// TIA Portal V17 export
// export: Created 2023-03-24T09:45:04.5136241Z, ExportSetting None, DisplayName Totally Integrated Automation Portal, DisplayVersion V17 Update 4, DisplayName TIA Portal Openness, DisplayVersion V17 Update 4, DisplayName TIA Portal Version Control Interface, DisplayVersion V17, DisplayName STEP 7 Professional, DisplayVersion V17 Update 4, DisplayName STEP 7 Safety, DisplayVersion V17, DisplayName WinCC Advanced / Unified PC, DisplayVersion V17 Update 4
FUNCTION "FC_DI" : Void   // FC12, LAD
TITLE = FC_DI
{ S7_Optimized_Access := 'FALSE' }
// Digital Input
// stored: SetENOAutomatically false
BEGIN

REGION Network 1: CONTROL VIA HW INTERFACE
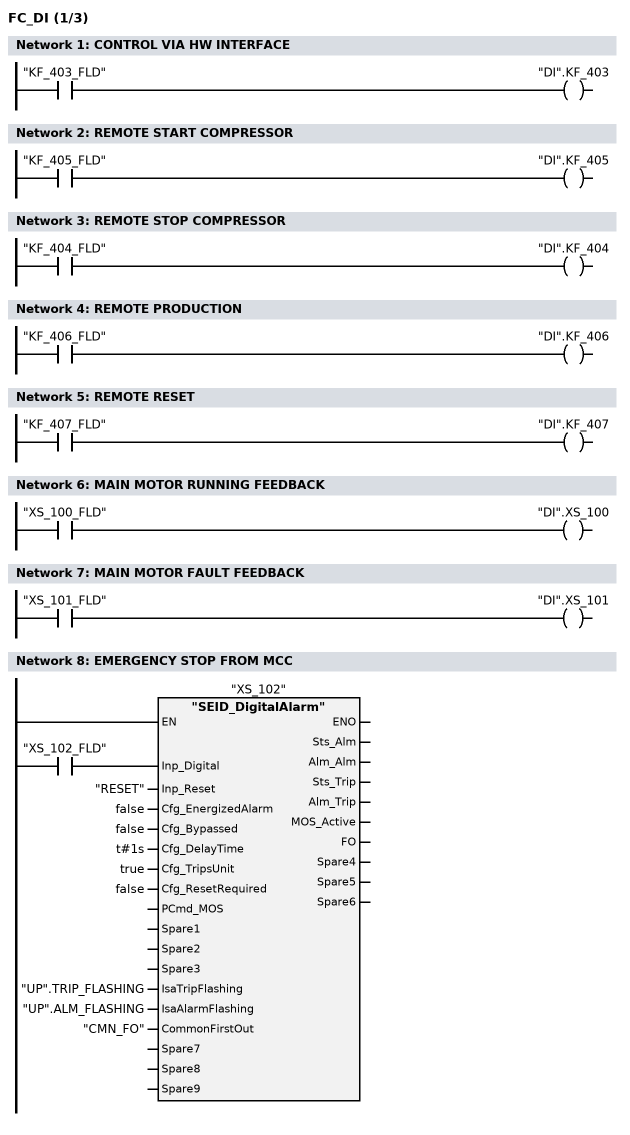
   RUNG wire#powerrail
      Contact( "KF_403_FLD" )
      Coil( "DI".KF_403 )
   END_RUNG
   // the same network as SCL:
   "DI".KF_403 := "KF_403_FLD";
END_REGION

REGION Network 2: REMOTE START COMPRESSOR
   RUNG wire#powerrail
      Contact( "KF_405_FLD" )
      Coil( "DI".KF_405 )
   END_RUNG
   // the same network as SCL:
   "DI".KF_405 := "KF_405_FLD";
END_REGION

REGION Network 3: REMOTE STOP COMPRESSOR
   RUNG wire#powerrail
      Contact( "KF_404_FLD" )
      Coil( "DI".KF_404 )
   END_RUNG
   // the same network as SCL:
   "DI".KF_404 := "KF_404_FLD";
END_REGION

REGION Network 4: REMOTE PRODUCTION
   RUNG wire#powerrail
      Contact( "KF_406_FLD" )
      Coil( "DI".KF_406 )
   END_RUNG
   // the same network as SCL:
   "DI".KF_406 := "KF_406_FLD";
END_REGION

REGION Network 5: REMOTE RESET
   RUNG wire#powerrail
      Contact( "KF_407_FLD" )
      Coil( "DI".KF_407 )
   END_RUNG
   // the same network as SCL:
   "DI".KF_407 := "KF_407_FLD";
END_REGION

REGION Network 6: MAIN MOTOR RUNNING FEEDBACK
   RUNG wire#powerrail
      Contact( "XS_100_FLD" )
      Coil( "DI".XS_100 )
   END_RUNG
   // the same network as SCL:
   "DI".XS_100 := "XS_100_FLD";
END_REGION

REGION Network 7: MAIN MOTOR FAULT FEEDBACK
   RUNG wire#powerrail
      Contact( "XS_101_FLD" )
      Coil( "DI".XS_101 )
   END_RUNG
   // the same network as SCL:
   "DI".XS_101 := "XS_101_FLD";
END_REGION

REGION Network 8: EMERGENCY STOP FROM MCC
   RUNG wire#powerrail
      "XS_102"(Inp_Digital := wire#w1, Inp_Reset := "RESET", Cfg_EnergizedAlarm := false, Cfg_Bypassed := false, Cfg_DelayTime := t#1s, Cfg_TripsUnit := true, Cfg_ResetRequired := false, PCmd_MOS :=, Spare1 :=, Spare2 :=, Spare3 :=, IsaTripFlashing := "UP".TRIP_FLASHING, IsaAlarmFlashing := "UP".ALM_FLASHING, CommonFirstOut := "CMN_FO", Spare7 :=, Spare8 :=, Spare9 :=, Sts_Alm =>, Alm_Alm =>, Sts_Trip =>, Alm_Trip =>, MOS_Active =>, FO =>, Spare4 =>, Spare5 =>, Spare6 =>)
   END_RUNG
   RUNG wire#powerrail
      Contact( "XS_102_FLD" )
   END_RUNG wire#w1
   // the same network as SCL:
   "XS_102"(Inp_Digital := "XS_102_FLD",   // "SEID_DigitalAlarm"
            Inp_Reset := "RESET",
            Cfg_EnergizedAlarm := false,
            Cfg_Bypassed := false,
            Cfg_DelayTime := t#1s,
            Cfg_TripsUnit := true,
            Cfg_ResetRequired := false,
            IsaTripFlashing := "UP".TRIP_FLASHING,
            IsaAlarmFlashing := "UP".ALM_FLASHING,
            CommonFirstOut := "CMN_FO");
END_REGION

REGION Network 9: HIGH TEMPERATURE FROM MCC
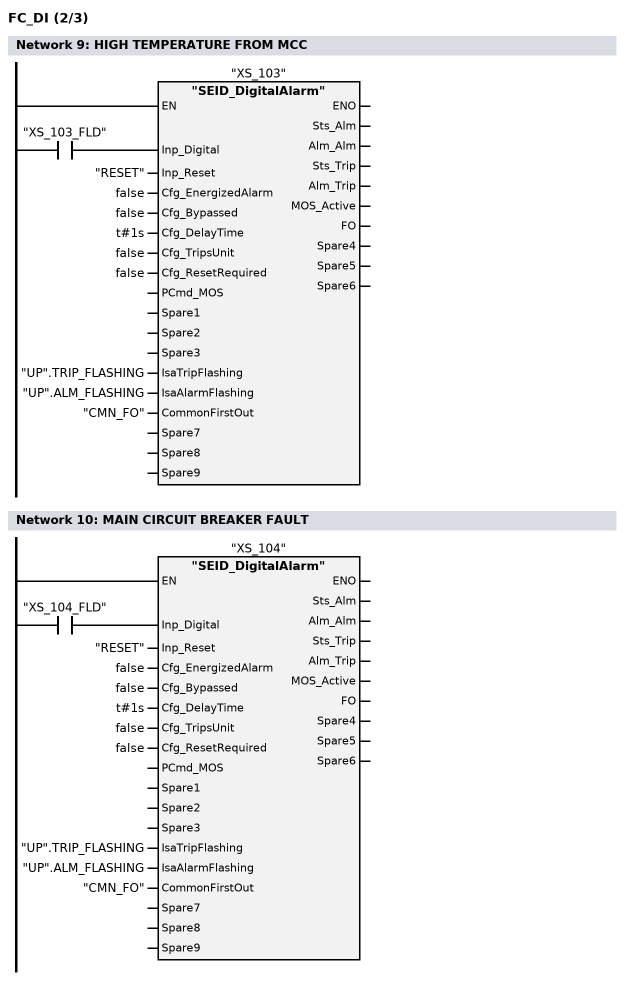
   RUNG wire#powerrail
      "XS_103"(Inp_Digital := wire#w1, Inp_Reset := "RESET", Cfg_EnergizedAlarm := false, Cfg_Bypassed := false, Cfg_DelayTime := t#1s, Cfg_TripsUnit := false, Cfg_ResetRequired := false, PCmd_MOS :=, Spare1 :=, Spare2 :=, Spare3 :=, IsaTripFlashing := "UP".TRIP_FLASHING, IsaAlarmFlashing := "UP".ALM_FLASHING, CommonFirstOut := "CMN_FO", Spare7 :=, Spare8 :=, Spare9 :=, Sts_Alm =>, Alm_Alm =>, Sts_Trip =>, Alm_Trip =>, MOS_Active =>, FO =>, Spare4 =>, Spare5 =>, Spare6 =>)
   END_RUNG
   RUNG wire#powerrail
      Contact( "XS_103_FLD" )
   END_RUNG wire#w1
   // the same network as SCL:
   "XS_103"(Inp_Digital := "XS_103_FLD",   // "SEID_DigitalAlarm"
            Inp_Reset := "RESET",
            Cfg_EnergizedAlarm := false,
            Cfg_Bypassed := false,
            Cfg_DelayTime := t#1s,
            Cfg_TripsUnit := false,
            Cfg_ResetRequired := false,
            IsaTripFlashing := "UP".TRIP_FLASHING,
            IsaAlarmFlashing := "UP".ALM_FLASHING,
            CommonFirstOut := "CMN_FO");
END_REGION

REGION Network 10: MAIN CIRCUIT BREAKER FAULT
   RUNG wire#powerrail
      "XS_104"(Inp_Digital := wire#w1, Inp_Reset := "RESET", Cfg_EnergizedAlarm := false, Cfg_Bypassed := false, Cfg_DelayTime := t#1s, Cfg_TripsUnit := false, Cfg_ResetRequired := false, PCmd_MOS :=, Spare1 :=, Spare2 :=, Spare3 :=, IsaTripFlashing := "UP".TRIP_FLASHING, IsaAlarmFlashing := "UP".ALM_FLASHING, CommonFirstOut := "CMN_FO", Spare7 :=, Spare8 :=, Spare9 :=, Sts_Alm =>, Alm_Alm =>, Sts_Trip =>, Alm_Trip =>, MOS_Active =>, FO =>, Spare4 =>, Spare5 =>, Spare6 =>)
   END_RUNG
   RUNG wire#powerrail
      Contact( "XS_104_FLD" )
   END_RUNG wire#w1
   // the same network as SCL:
   "XS_104"(Inp_Digital := "XS_104_FLD",   // "SEID_DigitalAlarm"
            Inp_Reset := "RESET",
            Cfg_EnergizedAlarm := false,
            Cfg_Bypassed := false,
            Cfg_DelayTime := t#1s,
            Cfg_TripsUnit := false,
            Cfg_ResetRequired := false,
            IsaTripFlashing := "UP".TRIP_FLASHING,
            IsaAlarmFlashing := "UP".ALM_FLASHING,
            CommonFirstOut := "CMN_FO");
END_REGION

REGION Network 11: UCP INTERNAL HIGH TEMPERATURE
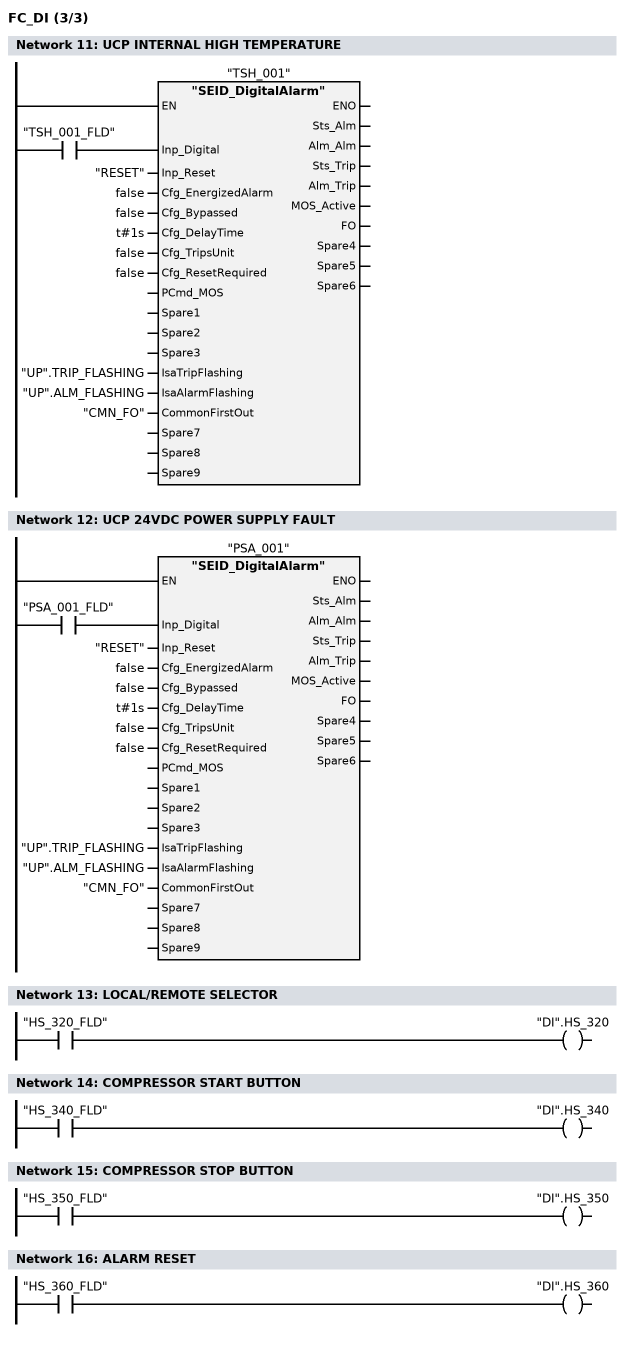
   RUNG wire#powerrail
      "TSH_001"(Inp_Digital := wire#w1, Inp_Reset := "RESET", Cfg_EnergizedAlarm := false, Cfg_Bypassed := false, Cfg_DelayTime := t#1s, Cfg_TripsUnit := false, Cfg_ResetRequired := false, PCmd_MOS :=, Spare1 :=, Spare2 :=, Spare3 :=, IsaTripFlashing := "UP".TRIP_FLASHING, IsaAlarmFlashing := "UP".ALM_FLASHING, CommonFirstOut := "CMN_FO", Spare7 :=, Spare8 :=, Spare9 :=, Sts_Alm =>, Alm_Alm =>, Sts_Trip =>, Alm_Trip =>, MOS_Active =>, FO =>, Spare4 =>, Spare5 =>, Spare6 =>)
   END_RUNG
   RUNG wire#powerrail
      Contact( "TSH_001_FLD" )
   END_RUNG wire#w1
   // the same network as SCL:
   "TSH_001"(Inp_Digital := "TSH_001_FLD",   // "SEID_DigitalAlarm"
             Inp_Reset := "RESET",
             Cfg_EnergizedAlarm := false,
             Cfg_Bypassed := false,
             Cfg_DelayTime := t#1s,
             Cfg_TripsUnit := false,
             Cfg_ResetRequired := false,
             IsaTripFlashing := "UP".TRIP_FLASHING,
             IsaAlarmFlashing := "UP".ALM_FLASHING,
             CommonFirstOut := "CMN_FO");
END_REGION

REGION Network 12: UCP 24VDC POWER SUPPLY FAULT
   RUNG wire#powerrail
      "PSA_001"(Inp_Digital := wire#w1, Inp_Reset := "RESET", Cfg_EnergizedAlarm := false, Cfg_Bypassed := false, Cfg_DelayTime := t#1s, Cfg_TripsUnit := false, Cfg_ResetRequired := false, PCmd_MOS :=, Spare1 :=, Spare2 :=, Spare3 :=, IsaTripFlashing := "UP".TRIP_FLASHING, IsaAlarmFlashing := "UP".ALM_FLASHING, CommonFirstOut := "CMN_FO", Spare7 :=, Spare8 :=, Spare9 :=, Sts_Alm =>, Alm_Alm =>, Sts_Trip =>, Alm_Trip =>, MOS_Active =>, FO =>, Spare4 =>, Spare5 =>, Spare6 =>)
   END_RUNG
   RUNG wire#powerrail
      Contact( "PSA_001_FLD" )
   END_RUNG wire#w1
   // the same network as SCL:
   "PSA_001"(Inp_Digital := "PSA_001_FLD",   // "SEID_DigitalAlarm"
             Inp_Reset := "RESET",
             Cfg_EnergizedAlarm := false,
             Cfg_Bypassed := false,
             Cfg_DelayTime := t#1s,
             Cfg_TripsUnit := false,
             Cfg_ResetRequired := false,
             IsaTripFlashing := "UP".TRIP_FLASHING,
             IsaAlarmFlashing := "UP".ALM_FLASHING,
             CommonFirstOut := "CMN_FO");
END_REGION

REGION Network 13: LOCAL/REMOTE SELECTOR
   RUNG wire#powerrail
      Contact( "HS_320_FLD" )
      Coil( "DI".HS_320 )
   END_RUNG
   // the same network as SCL:
   "DI".HS_320 := "HS_320_FLD";
END_REGION

REGION Network 14: COMPRESSOR START BUTTON
   RUNG wire#powerrail
      Contact( "HS_340_FLD" )
      Coil( "DI".HS_340 )
   END_RUNG
   // the same network as SCL:
   "DI".HS_340 := "HS_340_FLD";
END_REGION

REGION Network 15: COMPRESSOR STOP BUTTON
   RUNG wire#powerrail
      Contact( "HS_350_FLD" )
      Coil( "DI".HS_350 )
   END_RUNG
   // the same network as SCL:
   "DI".HS_350 := "HS_350_FLD";
END_REGION

REGION Network 16: ALARM RESET
   RUNG wire#powerrail
      Contact( "HS_360_FLD" )
      Coil( "DI".HS_360 )
   END_RUNG
   // the same network as SCL:
   "DI".HS_360 := "HS_360_FLD";
END_REGION
END_FUNCTION
